PROGRAM MAIN
VAR
	StringBuilderExample : CStringBuilderExample;
END_VAR

StringBuilderExample();

END_PROGRAM

(* stored: Version 1.1.0.1, ProductVersion 3.1.4024.13
   POU MAIN: Id {1545be35-79c0-49e0-9439-af023340e6dc}, SpecialFunc None *)
